FUNCTION_BLOCK MyCalculatorTestSuite
VAR
	_DivideByZeroTest : DivideByZeroTest;
END_VAR

_DivideByZeroTest.RunTest();

END_FUNCTION_BLOCK

(* stored: Version 1.1.0.1, ProductVersion 3.1.4024.13
   POU MyCalculatorTestSuite: Id {978c53fb-e274-41e2-85d0-07d6e20d6a57}, SpecialFunc None *)
